(* Logix 5000 project; controller cal1615 1756-L62 rev 20.11; software revision 20.05; part 10 of 81 *)
(* tags used below, declared in another part *)
   FAULT : BOOL;   // Fault AFI
   HMI : BOOL;   // AFI HMI
   p01_dint_to_hmi : DINT[16];   // System Dint to HMI
   p01_int_from_oxidizer : INT[10];   // System Oxidizer Int from Oxidizer
   p01_param_master_jog_speed : REAL;   // Machine Parameter Master Jog Speed
   p01_real_to_hmi : REAL[112];   // System Real to HMI
   p01r01 : routine;
   p01r02 : routine;   // System Misc Control
   p01r05 : routine;   // System Dint to HMI
   p01r05_timer_warning : TIMER[4];   // System Dint to HMI Warning Delay
   p01r06 : routine;   // System Real to HMI
   p01r06_timer_fault : TIMER[4];   // System Real to HMI Fault Delay
   p01r06_timer_warning : TIMER[4];   // System Real to HMI Warning Delay
   p01r07 : routine;   // System Alarms
   p01r07_timer_fault : TIMER[4];   // System Alarms Fault Delay
   p01r07_timer_warning : TIMER[4];   // System Alarms Warning Delay
   p01r08 : routine;   // System Warnings
   p01r08_timer_fault : TIMER[4];   // System Warnings Fault Delay
   p01r08_timer_warning : TIMER[4];   // System Warnings Warning Delay
   p01r09 : routine;   // System Modes
   p01r09_pb_global_reset : BOOL;   // System Modes PB: Global Fault Reset
   p01r12_master_ramped_speed : REAL;   // System Line Accel Decel Control Master Ramped Speed
   p01r14 : routine;
   p01r14_oxidizer_mass_flow : REAL;   // System Oxidizer Oxidizer Mass Flow [SCFM]
   p20r18_index_complete : BOOL;   // Letoff Letoff Turret VFD Index Complete
(* P01_System, continued *)

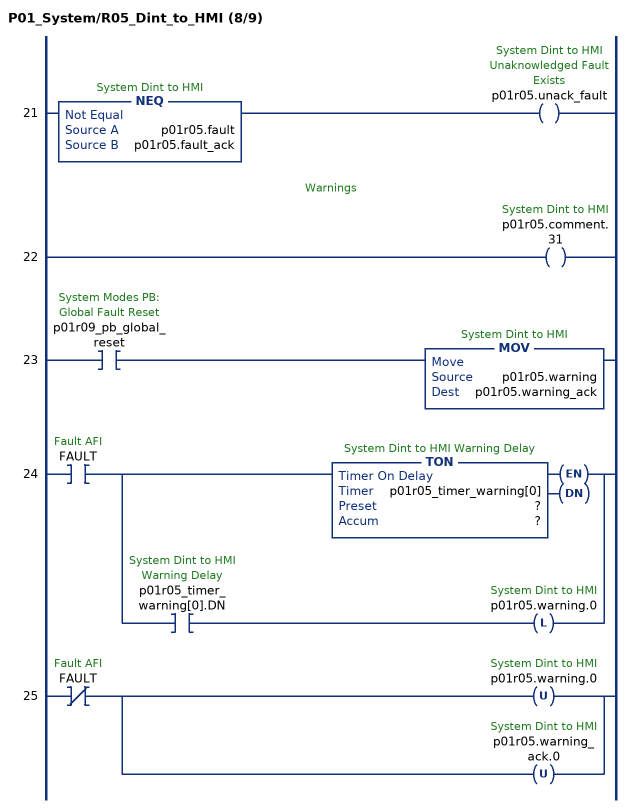
   [picture p91: P01_System/R05_Dint_to_HMI rungs 21-25]
   21: NEQ(p01r05.fault,p01r05.fault_ack)OTE(p01r05.unack_fault);
   // Warnings
   22: OTE(p01r05.comment.31);
   23: XIC(p01r09_pb_global_reset)MOV(p01r05.warning,p01r05.warning_ack);
   24: XIC(FAULT)[TON(p01r05_timer_warning[0],?,?) ,XIC(p01r05_timer_warning[0].DN) OTL(p01r05.warning.0) ];
   25: XIO(FAULT)[OTU(p01r05.warning.0) ,OTU(p01r05.warning_ack.0) ];
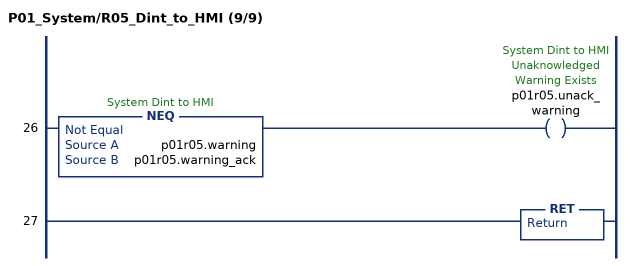
   26: NEQ(p01r05.warning,p01r05.warning_ack)OTE(p01r05.unack_warning);
   27: RET();
END_ROUTINE

ROUTINE R06_Real_to_HMI   (* ladder *)
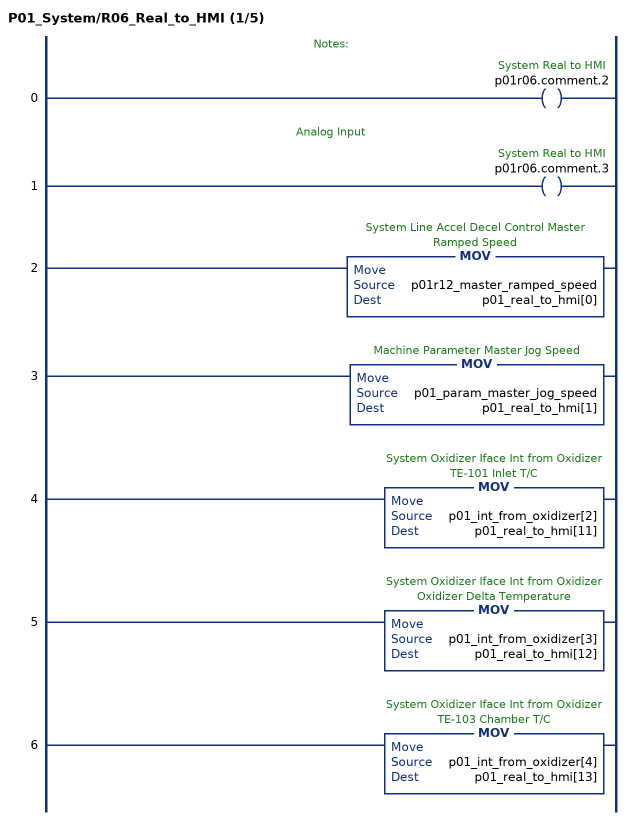
   // Notes:
   0: OTE(p01r06.comment.2);
   // Analog Input
   1: OTE(p01r06.comment.3);
   2: MOV(p01r12_master_ramped_speed,p01_real_to_hmi[0]);
   3: MOV(p01_param_master_jog_speed,p01_real_to_hmi[1]);
   4: MOV(p01_int_from_oxidizer[2],p01_real_to_hmi[11]);
   5: MOV(p01_int_from_oxidizer[3],p01_real_to_hmi[12]);
   6: MOV(p01_int_from_oxidizer[4],p01_real_to_hmi[13]);
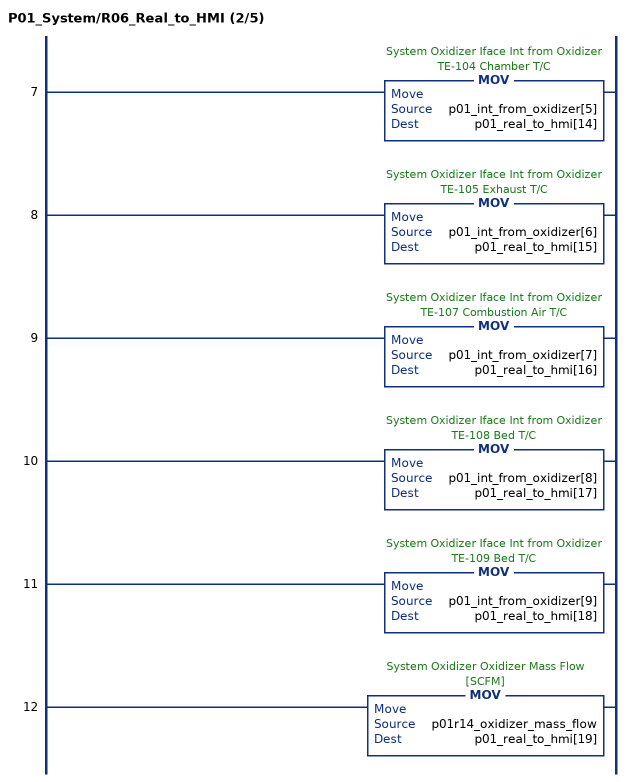
   7: MOV(p01_int_from_oxidizer[5],p01_real_to_hmi[14]);
   8: MOV(p01_int_from_oxidizer[6],p01_real_to_hmi[15]);
   9: MOV(p01_int_from_oxidizer[7],p01_real_to_hmi[16]);
   10: MOV(p01_int_from_oxidizer[8],p01_real_to_hmi[17]);
   11: MOV(p01_int_from_oxidizer[9],p01_real_to_hmi[18]);
   12: MOV(p01r14_oxidizer_mass_flow,p01_real_to_hmi[19]);
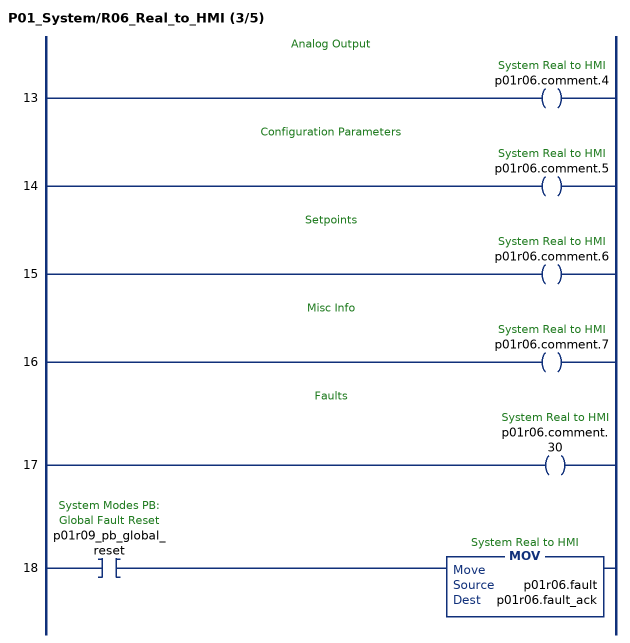
   // Analog Output
   13: OTE(p01r06.comment.4);
   // Configuration Parameters
   14: OTE(p01r06.comment.5);
   // Setpoints
   15: OTE(p01r06.comment.6);
   // Misc Info
   16: OTE(p01r06.comment.7);
   // Faults
   17: OTE(p01r06.comment.30);
   18: XIC(p01r09_pb_global_reset)MOV(p01r06.fault,p01r06.fault_ack);
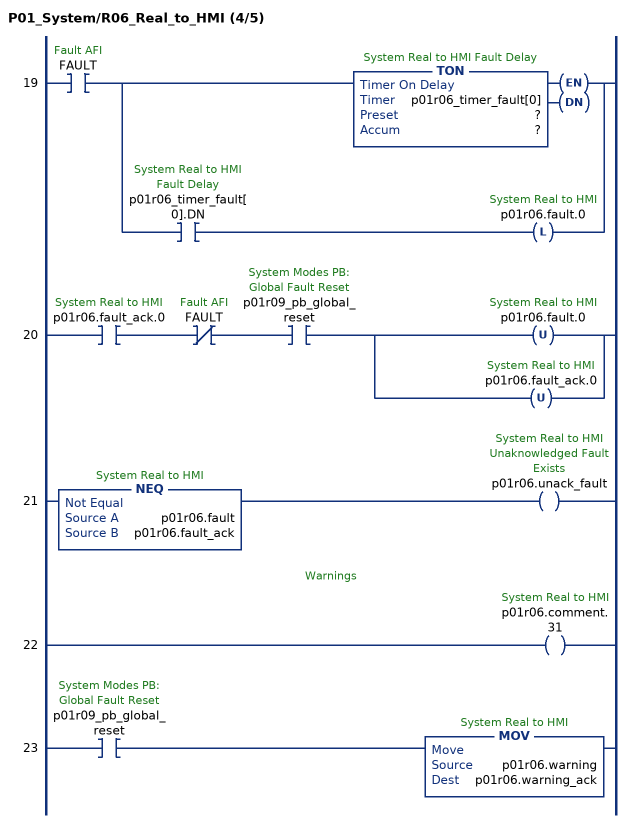
   19: XIC(FAULT)[TON(p01r06_timer_fault[0],?,?) ,XIC(p01r06_timer_fault[0].DN) OTL(p01r06.fault.0) ];
   20: XIC(p01r06.fault_ack.0)XIO(FAULT)XIC(p01r09_pb_global_reset)[OTU(p01r06.fault.0) ,OTU(p01r06.fault_ack.0) ];
   21: NEQ(p01r06.fault,p01r06.fault_ack)OTE(p01r06.unack_fault);
   // Warnings
   22: OTE(p01r06.comment.31);
   23: XIC(p01r09_pb_global_reset)MOV(p01r06.warning,p01r06.warning_ack);
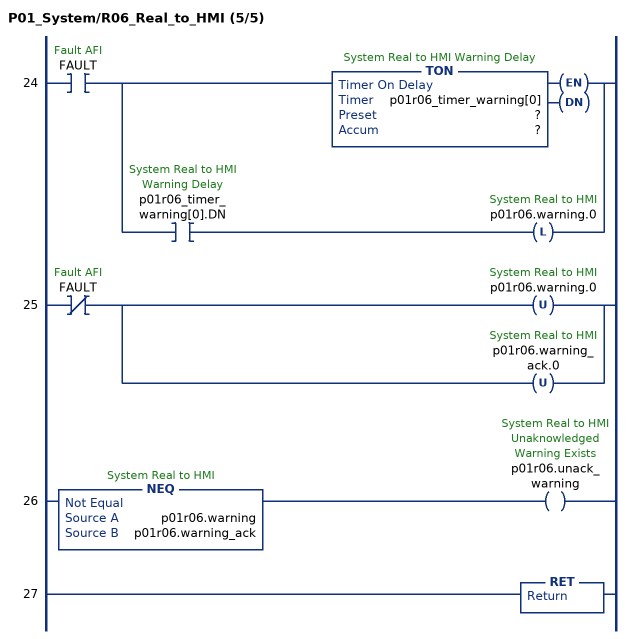
   24: XIC(FAULT)[TON(p01r06_timer_warning[0],?,?) ,XIC(p01r06_timer_warning[0].DN) OTL(p01r06.warning.0) ];
   25: XIO(FAULT)[OTU(p01r06.warning.0) ,OTU(p01r06.warning_ack.0) ];
   26: NEQ(p01r06.warning,p01r06.warning_ack)OTE(p01r06.unack_warning);
   27: RET();
END_ROUTINE

ROUTINE R07_Alarms   (* ladder *)
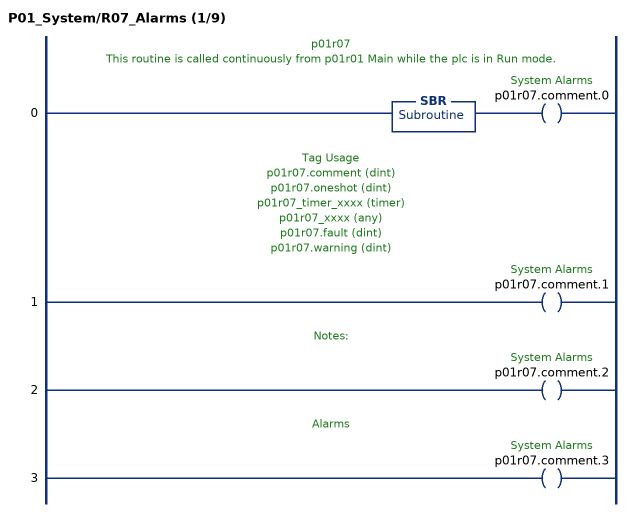
   // p01r07
   // This routine is called continuously from p01r01 Main while the plc is in Run mode.
   0: SBR()OTE(p01r07.comment.0);
   // Tag Usage
   // p01r07.comment (dint)
   // p01r07.oneshot (dint)
   // p01r07_timer_xxxx (timer)
   // p01r07_xxxx (any)
   // p01r07.fault (dint)
   // p01r07.warning (dint)
   1: OTE(p01r07.comment.1);
   // Notes:
   2: OTE(p01r07.comment.2);
   // Alarms
   3: OTE(p01r07.comment.3);
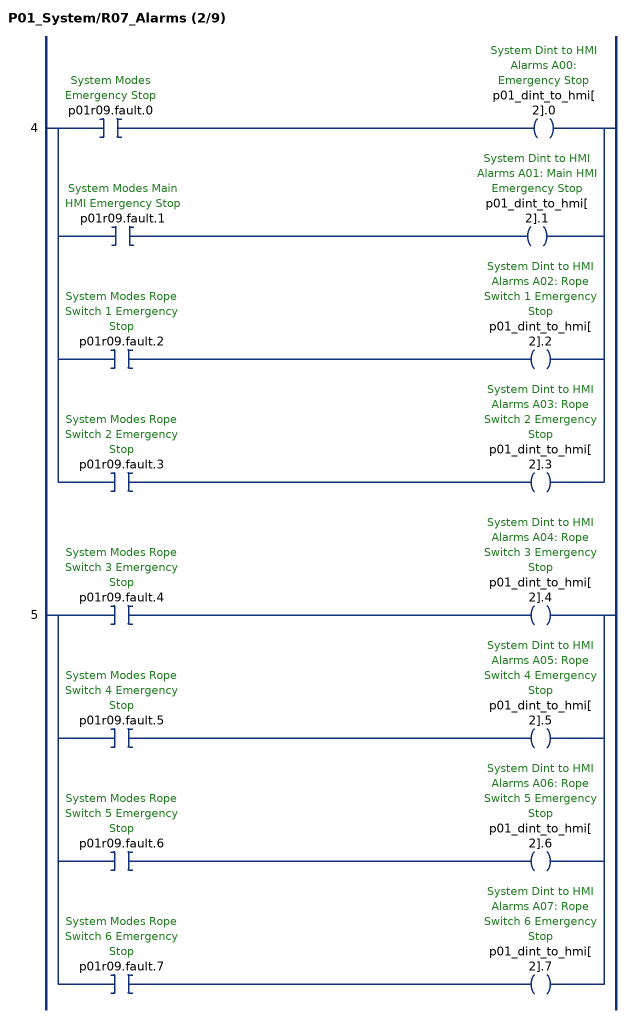
   4: [XIC(p01r09.fault.0) OTE(p01_dint_to_hmi[2].0) ,XIC(p01r09.fault.1) OTE(p01_dint_to_hmi[2].1) ,XIC(p01r09.fault.2) OTE(p01_dint_to_hmi[2].2) ,XIC(p01r09.fault.3) OTE(p01_dint_to_hmi[2].3) ];
   5: [XIC(p01r09.fault.4) OTE(p01_dint_to_hmi[2].4) ,XIC(p01r09.fault.5) OTE(p01_dint_to_hmi[2].5) ,XIC(p01r09.fault.6) OTE(p01_dint_to_hmi[2].6) ,XIC(p01r09.fault.7) OTE(p01_dint_to_hmi[2].7) ];
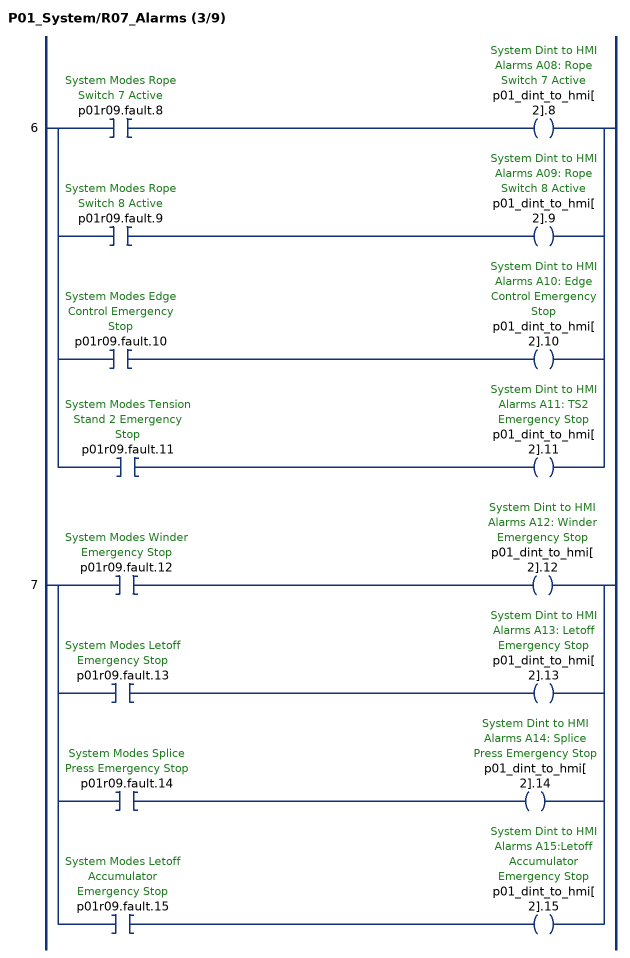
   6: [XIC(p01r09.fault.8) OTE(p01_dint_to_hmi[2].8) ,XIC(p01r09.fault.9) OTE(p01_dint_to_hmi[2].9) ,XIC(p01r09.fault.10) OTE(p01_dint_to_hmi[2].10) ,XIC(p01r09.fault.11) OTE(p01_dint_to_hmi[2].11) ];
   7: [XIC(p01r09.fault.12) OTE(p01_dint_to_hmi[2].12) ,XIC(p01r09.fault.13) OTE(p01_dint_to_hmi[2].13) ,XIC(p01r09.fault.14) OTE(p01_dint_to_hmi[2].14) ,XIC(p01r09.fault.15) OTE(p01_dint_to_hmi[2].15) ];
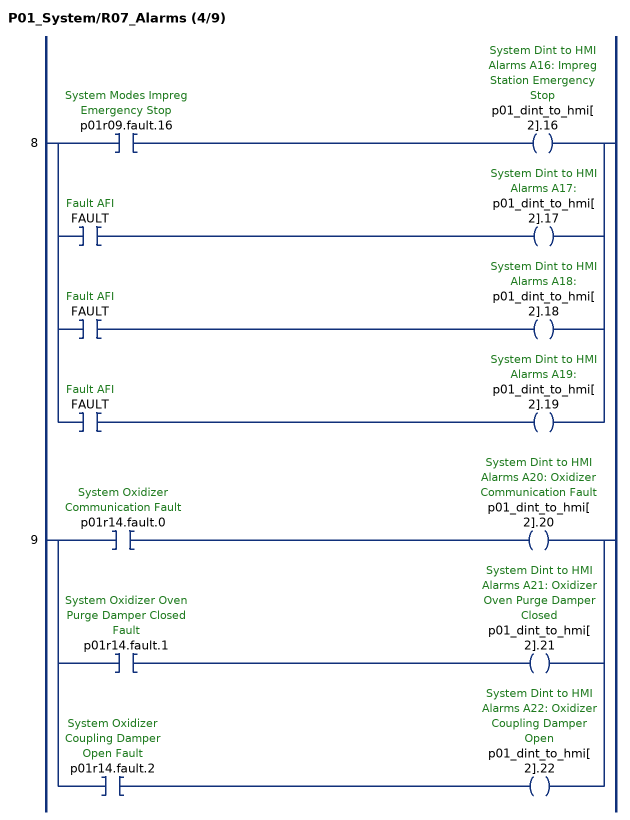
   8: [XIC(p01r09.fault.16) OTE(p01_dint_to_hmi[2].16) ,XIC(FAULT) OTE(p01_dint_to_hmi[2].17) ,XIC(FAULT) OTE(p01_dint_to_hmi[2].18) ,XIC(FAULT) OTE(p01_dint_to_hmi[2].19) ];
   9: [XIC(p01r14.fault.0) OTE(p01_dint_to_hmi[2].20) ,XIC(p01r14.fault.1) OTE(p01_dint_to_hmi[2].21) ,XIC(p01r14.fault.2) OTE(p01_dint_to_hmi[2].22) ];
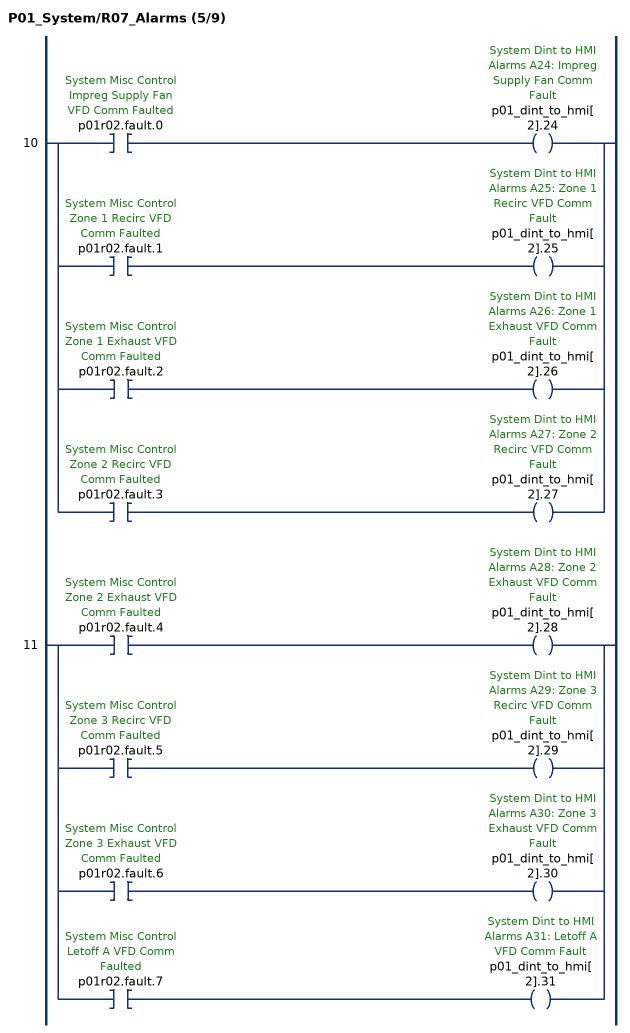
   10: [XIC(p01r02.fault.0) OTE(p01_dint_to_hmi[2].24) ,XIC(p01r02.fault.1) OTE(p01_dint_to_hmi[2].25) ,XIC(p01r02.fault.2) OTE(p01_dint_to_hmi[2].26) ,XIC(p01r02.fault.3) OTE(p01_dint_to_hmi[2].27) ];
   11: [XIC(p01r02.fault.4) OTE(p01_dint_to_hmi[2].28) ,XIC(p01r02.fault.5) OTE(p01_dint_to_hmi[2].29) ,XIC(p01r02.fault.6) OTE(p01_dint_to_hmi[2].30) ,XIC(p01r02.fault.7) OTE(p01_dint_to_hmi[2].31) ];
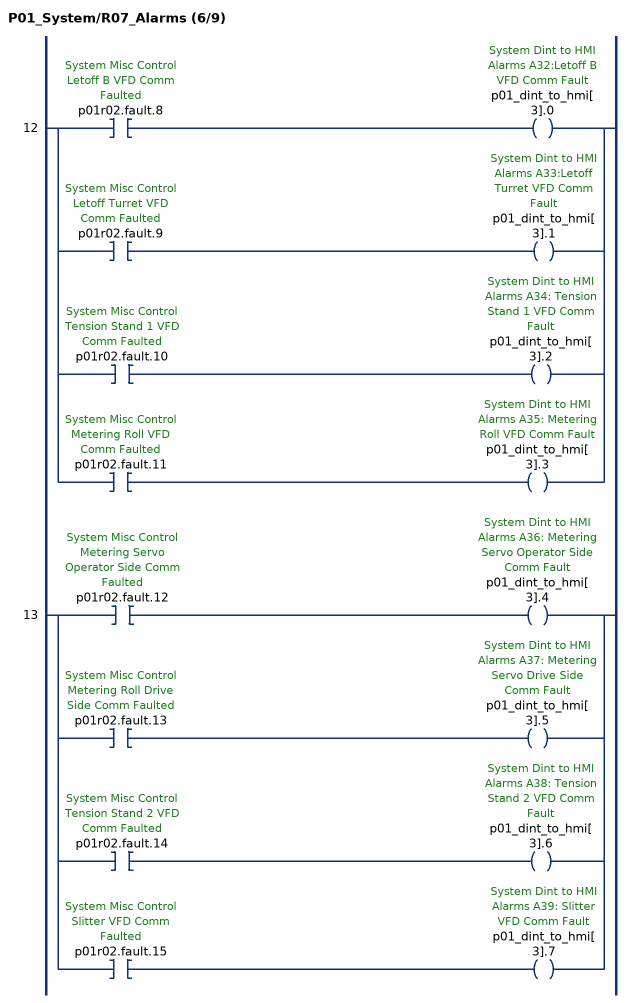
   12: [XIC(p01r02.fault.8) OTE(p01_dint_to_hmi[3].0) ,XIC(p01r02.fault.9) OTE(p01_dint_to_hmi[3].1) ,XIC(p01r02.fault.10) OTE(p01_dint_to_hmi[3].2) ,XIC(p01r02.fault.11) OTE(p01_dint_to_hmi[3].3) ];
   13: [XIC(p01r02.fault.12) OTE(p01_dint_to_hmi[3].4) ,XIC(p01r02.fault.13) OTE(p01_dint_to_hmi[3].5) ,XIC(p01r02.fault.14) OTE(p01_dint_to_hmi[3].6) ,XIC(p01r02.fault.15) OTE(p01_dint_to_hmi[3].7) ];
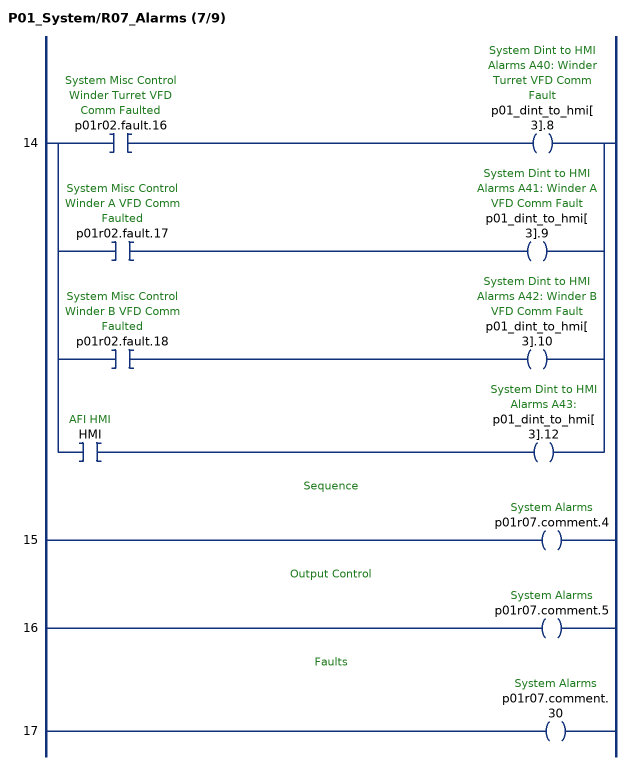
   14: [XIC(p01r02.fault.16) OTE(p01_dint_to_hmi[3].8) ,XIC(p01r02.fault.17) OTE(p01_dint_to_hmi[3].9) ,XIC(p01r02.fault.18) OTE(p01_dint_to_hmi[3].10) ,XIC(HMI) OTE(p01_dint_to_hmi[3].12) ];
   // Sequence
   15: OTE(p01r07.comment.4);
   // Output Control
   16: OTE(p01r07.comment.5);
   // Faults
   17: OTE(p01r07.comment.30);
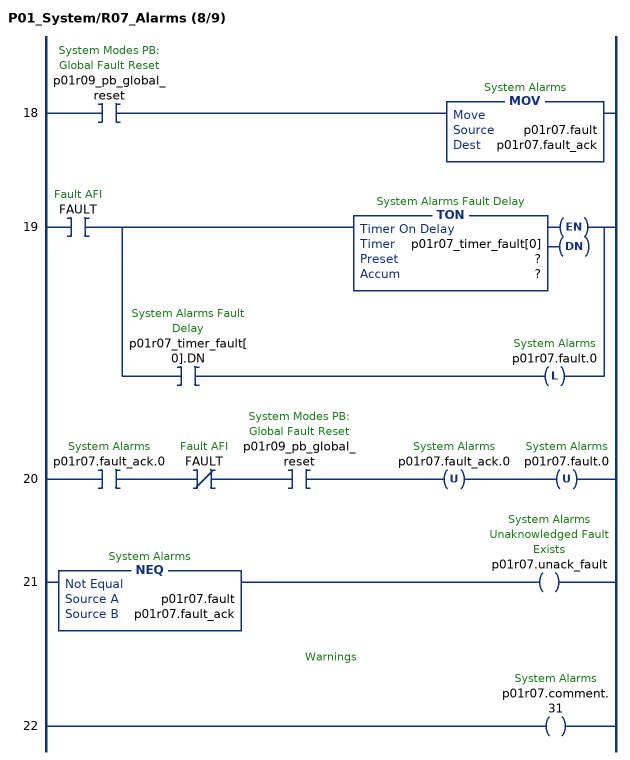
   18: XIC(p01r09_pb_global_reset)MOV(p01r07.fault,p01r07.fault_ack);
   19: XIC(FAULT)[TON(p01r07_timer_fault[0],?,?) ,XIC(p01r07_timer_fault[0].DN) OTL(p01r07.fault.0) ];
   20: XIC(p01r07.fault_ack.0)XIO(FAULT)XIC(p01r09_pb_global_reset)OTU(p01r07.fault_ack.0)OTU(p01r07.fault.0);
   21: NEQ(p01r07.fault,p01r07.fault_ack)OTE(p01r07.unack_fault);
   // Warnings
   22: OTE(p01r07.comment.31);
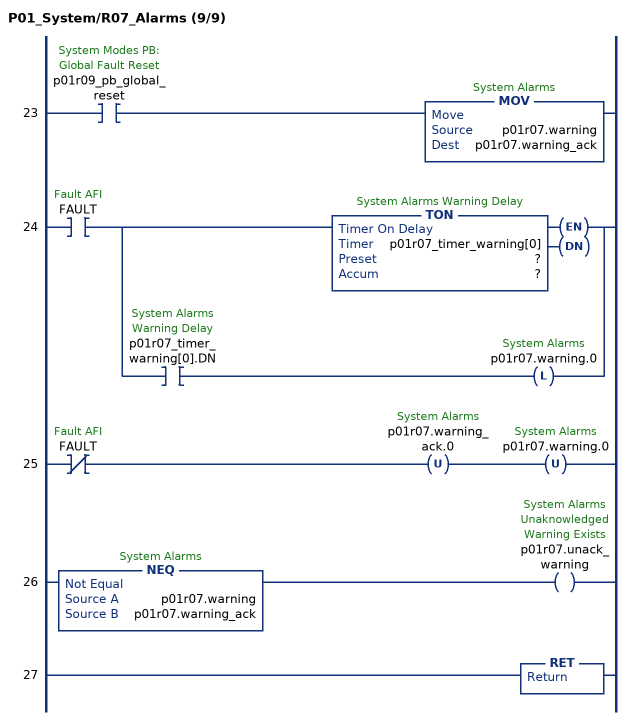
   23: XIC(p01r09_pb_global_reset)MOV(p01r07.warning,p01r07.warning_ack);
   24: XIC(FAULT)[TON(p01r07_timer_warning[0],?,?) ,XIC(p01r07_timer_warning[0].DN) OTL(p01r07.warning.0) ];
   25: XIO(FAULT)OTU(p01r07.warning_ack.0)OTU(p01r07.warning.0);
   26: NEQ(p01r07.warning,p01r07.warning_ack)OTE(p01r07.unack_warning);
   27: RET();
END_ROUTINE

ROUTINE R08_Warnings   (* ladder *)
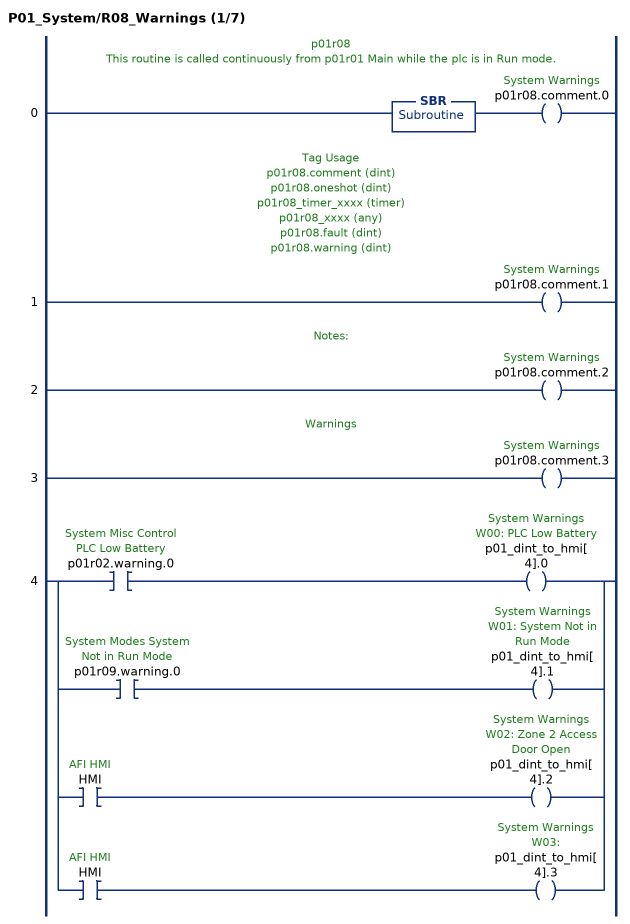
   // p01r08
   // This routine is called continuously from p01r01 Main while the plc is in Run mode.
   0: SBR()OTE(p01r08.comment.0);
   // Tag Usage
   // p01r08.comment (dint)
   // p01r08.oneshot (dint)
   // p01r08_timer_xxxx (timer)
   // p01r08_xxxx (any)
   // p01r08.fault (dint)
   // p01r08.warning (dint)
   1: OTE(p01r08.comment.1);
   // Notes:
   2: OTE(p01r08.comment.2);
   // Warnings
   3: OTE(p01r08.comment.3);
   4: [XIC(p01r02.warning.0) OTE(p01_dint_to_hmi[4].0) ,XIC(p01r09.warning.0) OTE(p01_dint_to_hmi[4].1) ,XIC(HMI) OTE(p01_dint_to_hmi[4].2) ,XIC(HMI) OTE(p01_dint_to_hmi[4].3) ];
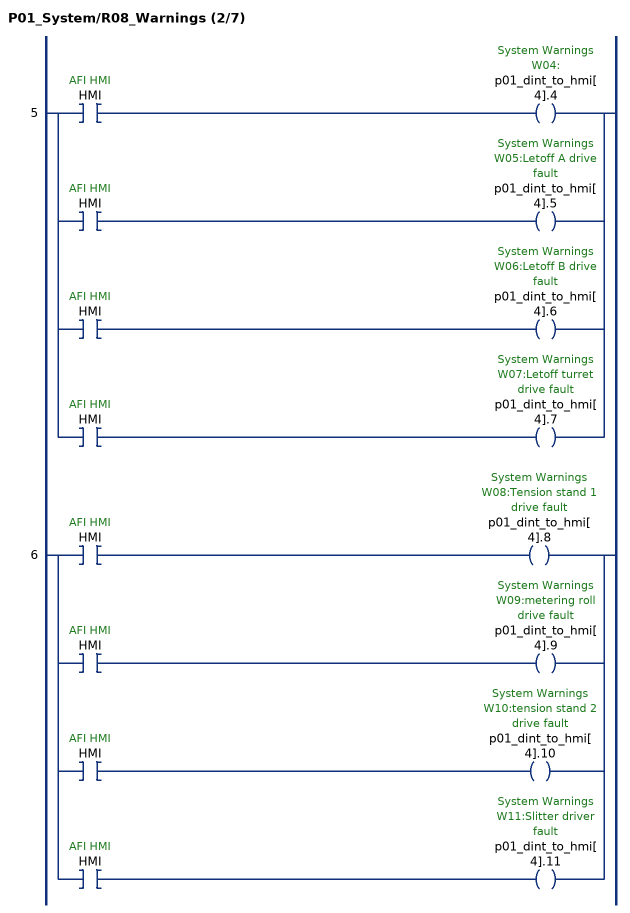
   5: [XIC(HMI) OTE(p01_dint_to_hmi[4].4) ,XIC(HMI) OTE(p01_dint_to_hmi[4].5) ,XIC(HMI) OTE(p01_dint_to_hmi[4].6) ,XIC(HMI) OTE(p01_dint_to_hmi[4].7) ];
   6: [XIC(HMI) OTE(p01_dint_to_hmi[4].8) ,XIC(HMI) OTE(p01_dint_to_hmi[4].9) ,XIC(HMI) OTE(p01_dint_to_hmi[4].10) ,XIC(HMI) OTE(p01_dint_to_hmi[4].11) ];
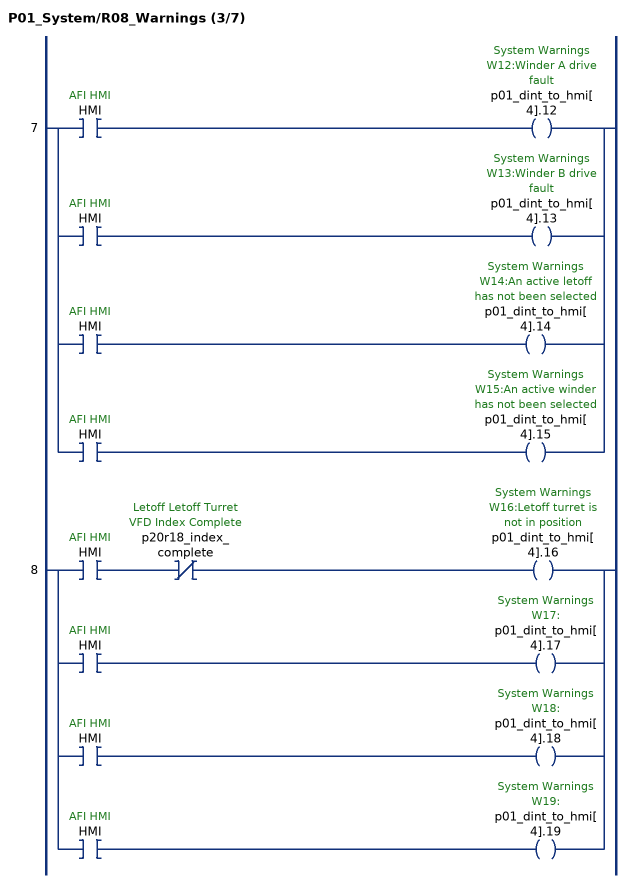
   7: [XIC(HMI) OTE(p01_dint_to_hmi[4].12) ,XIC(HMI) OTE(p01_dint_to_hmi[4].13) ,XIC(HMI) OTE(p01_dint_to_hmi[4].14) ,XIC(HMI) OTE(p01_dint_to_hmi[4].15) ];
   8: [XIC(HMI) XIO(p20r18_index_complete) OTE(p01_dint_to_hmi[4].16) ,XIC(HMI) OTE(p01_dint_to_hmi[4].17) ,XIC(HMI) OTE(p01_dint_to_hmi[4].18) ,XIC(HMI) OTE(p01_dint_to_hmi[4].19) ];
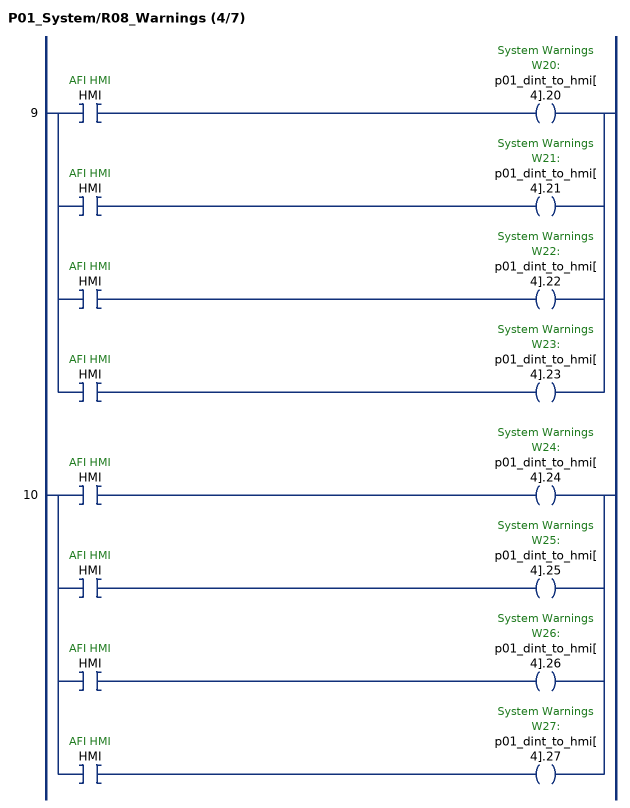
   9: [XIC(HMI) OTE(p01_dint_to_hmi[4].20) ,XIC(HMI) OTE(p01_dint_to_hmi[4].21) ,XIC(HMI) OTE(p01_dint_to_hmi[4].22) ,XIC(HMI) OTE(p01_dint_to_hmi[4].23) ];
   10: [XIC(HMI) OTE(p01_dint_to_hmi[4].24) ,XIC(HMI) OTE(p01_dint_to_hmi[4].25) ,XIC(HMI) OTE(p01_dint_to_hmi[4].26) ,XIC(HMI) OTE(p01_dint_to_hmi[4].27) ];
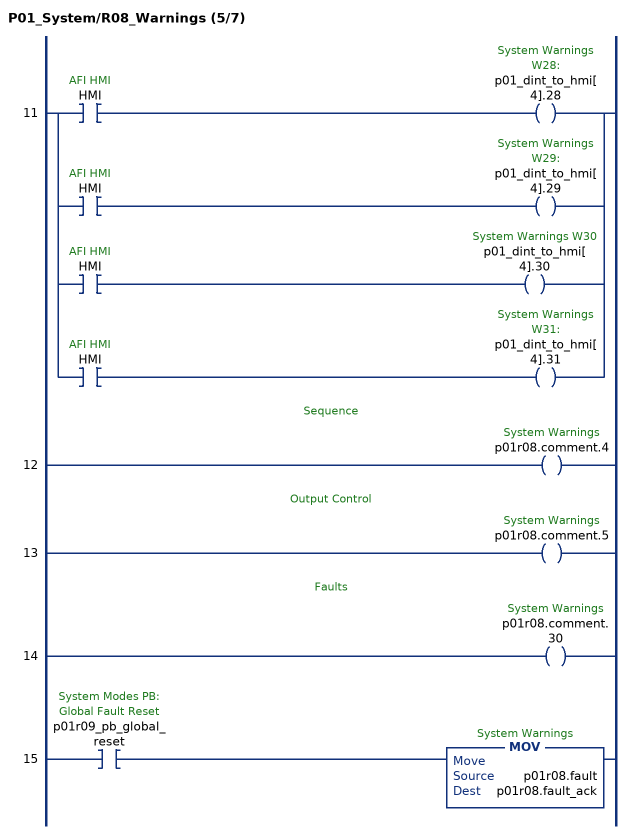
   11: [XIC(HMI) OTE(p01_dint_to_hmi[4].28) ,XIC(HMI) OTE(p01_dint_to_hmi[4].29) ,XIC(HMI) OTE(p01_dint_to_hmi[4].30) ,XIC(HMI) OTE(p01_dint_to_hmi[4].31) ];
   // Sequence
   12: OTE(p01r08.comment.4);
   // Output Control
   13: OTE(p01r08.comment.5);
   // Faults
   14: OTE(p01r08.comment.30);
   15: XIC(p01r09_pb_global_reset)MOV(p01r08.fault,p01r08.fault_ack);
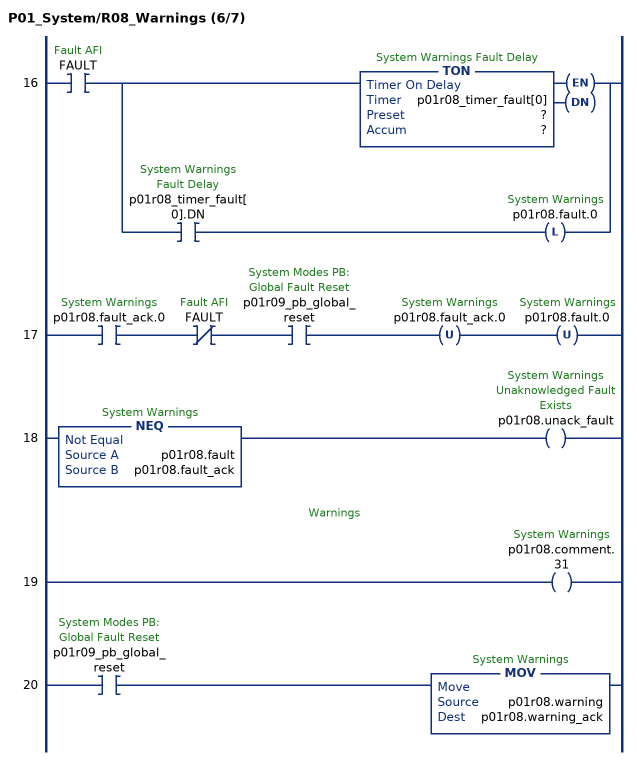
   16: XIC(FAULT)[TON(p01r08_timer_fault[0],?,?) ,XIC(p01r08_timer_fault[0].DN) OTL(p01r08.fault.0) ];
   17: XIC(p01r08.fault_ack.0)XIO(FAULT)XIC(p01r09_pb_global_reset)OTU(p01r08.fault_ack.0)OTU(p01r08.fault.0);
   18: NEQ(p01r08.fault,p01r08.fault_ack)OTE(p01r08.unack_fault);
   // Warnings
   19: OTE(p01r08.comment.31);
   20: XIC(p01r09_pb_global_reset)MOV(p01r08.warning,p01r08.warning_ack);
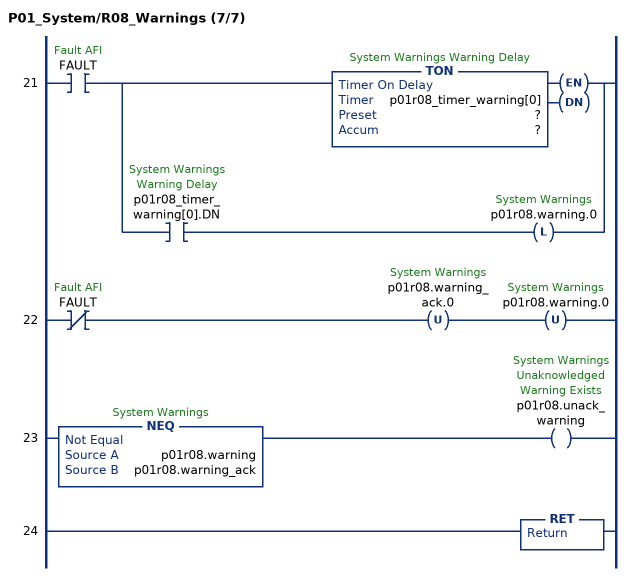
   21: XIC(FAULT)[TON(p01r08_timer_warning[0],?,?) ,XIC(p01r08_timer_warning[0].DN) OTL(p01r08.warning.0) ];
   22: XIO(FAULT)OTU(p01r08.warning_ack.0)OTU(p01r08.warning.0);
   23: NEQ(p01r08.warning,p01r08.warning_ack)OTE(p01r08.unack_warning);
   24: RET();
END_ROUTINE
